# EPICS substitutions: ek9000App/Db/EL1382_mbbiDirect.substitutions
file EL1382.template
{       pattern
        {
                TERMINAL,

        }
        {
        }
}
